{attribute 'qualified_only'}
VAR_GLOBAL CONSTANT
	COMMAND_QUEUE_BUFFER_SIZE :UINT := 10;
	MAX_OBSERVATION_SDO :UINT := 100;
END_VAR

(* stored: Version 1.1.0.1, ProductVersion 3.1.4024.12
   GVL ParameterList: Id {87829346-087a-4326-a2ca-1fe5098422eb}, ParameterList True *)
